{attribute 'qualified_only'}
{attribute 'strict'}

//TYPE PizzaType :
//(
//	mozorela := 1,
//	tuna := 2

//);
//END_TYPE

(* stored: Version 1.1.0.1, ProductVersion 3.1.4022.6
   EnumerationTextList PizzaType: Id {f48fa107-516d-4cc3-8088-fc1179f6760c} *)
